(* CoDeSys 2.3.9.47 project: ATS_P8.pro *)
(* Libraries: STANDARD.LIB 5.6.98 12:03:02 *)

(* Task configuration *)
TASK Standard (PRIORITY := 0, INTERVAL := T#10ms);
	MAIN
END_TASK

(* Global variable list: Global_Variables *)
VAR_GLOBAL
(*Analog Input*)
intUSS  	AT%I* : INT;
(*Analog Output*)
analogOut	AT%Q* : INT;
END_VAR

(* POU MAIN, ST *)
PROGRAM MAIN
VAR
n		: INT := 8;	(*Quantification*)
v_max	: INT := 10; (*Analog Display Range*)
voltUSS	:REAL := 0; (*Sensor Voltage*)
END_VAR
(*Calculate Sensor Voltage *)

(*Output Analog Signal*)
analogOut := REAL_TO_INT();
END_PROGRAM
